PROGRAM P_Unit_Tests
VAR
	fbFoo_Tests		:	FB_Foo_Tests;	
END_VAR

fbFoo_Tests();

END_PROGRAM

(* stored: Version 1.1.0.1, ProductVersion 3.1.4022.7
   POU P_Unit_Tests: Id {08c39198-6e34-4947-81d5-6830d7c1050c}, SpecialFunc None *)
